// TIA Portal project "Aufgabe_2_001_mCopilot" (V20)

(* hardware
DEVICE "S7-1200 G2 station_1"  S7-1200 G2 Station
   slot 0: "Rack_0"  S71200G2 Rack  Rack  V1.0
   slot 1: "PLC_1"  CPU 1212C DC/DC/DC  6ES7 212-1AG50-0XB0  V1.0
*)

// ===== PLC "PLC_1"  CPU 1212C DC/DC/DC =====

VAR_GLOBAL   // PLC tag table "Default tag table"
   "S1" AT %I0.0 : Bool;
   "S2" AT %I0.1 : Bool;
   "S3" AT %I0.2 : Bool;
   "S4" AT %I0.3 : Bool;
   "M1" AT %Q0.0 : Bool;
   "M2" AT %Q0.1 : Bool;
   "M3" AT %Q0.2 : Bool;
   "M4" AT %Q0.3 : Bool;
   "Clock_Byte" AT %MB0 : Byte;
   "Clock_10Hz" AT %M0.0 : Bool;
   "Clock_5Hz" AT %M0.1 : Bool;
   "Clock_2.5Hz" AT %M0.2 : Bool;
   "Clock_2Hz" AT %M0.3 : Bool;
   "Clock_1.25Hz" AT %M0.4 : Bool;
   "Clock_1Hz" AT %M0.5 : Bool;
   "Clock_0.625Hz" AT %M0.6 : Bool;
   "Clock_0.5Hz" AT %M0.7 : Bool;
   "VarOverflow" AT %Q0.4 : Bool;
END_VAR

VAR_GLOBAL CONSTANT   // PLC tag table "Default tag table"
   "WARNING_THRESHOLD" : Int := 100;
END_VAR

// folder: Instances

DATA_BLOCK "InstFB_BaggageCarousel"   // DB1
{ S7_Optimized_Access := 'TRUE' }
VERSION : 0.1
// stored: InstanceOfName FB_BaggageCarousel
"FB_BaggageCarousel"
BEGIN
END_DATA_BLOCK

// folder: System blocks/Program resources

DATA_BLOCK "InstTickCunt"   // DB2
{ S7_Optimized_Access := 'TRUE' }
AUTHOR : SIMATIC
FAMILY : IEC
NAME : DCNTR
VERSION : 1.2
// stored: InstanceOfName IEC_DCOUNTER
"IEC_DCOUNTER"
BEGIN
END_DATA_BLOCK

// folder: (top level)

FUNCTION_BLOCK "FB_BaggageCarousel"   // FB21, SCL
{ S7_Optimized_Access := 'TRUE' }
VERSION : 0.1
   VAR_INPUT
      infeedConveyorS1 : Bool;   // S1
      infeedConveyorS2 : Bool;   // S2
      infeedConveyorS3 : Bool;   // S3
      circularConveyorS4 : Bool;   // S4
      clockInput : DInt;
   END_VAR
   VAR_OUTPUT
      infeedCoveyorM1 : Bool;   // M1
      infeedCoveyorM2 : Bool;   // M2
      infeedCoveyorM3 : Bool;   // M3
      circularConveyorM4 : Bool;   // M4
      clockReset : Bool;
   END_VAR
   VAR
      statInfeedConveyorM3Run : Bool;
      statInfeedConveyorM2Run : Bool;
      statInfeedConveyorM1Run : Bool;
      instInfeedPointAllowWindow : TP_TIME;
      instInfeedPointMonitor : TON_TIME;
      statClockMem : Array[0..100] of DInt;
      statClockCurrent : DInt;
      statInfeedConveyorS1BaggageDetected : Bool;   // S1
      statInfeedConveyorS2BaggageDetected : Bool;   // S2
      statInfeedConveyorS3BaggageDetected : Bool;   // S3
      statCircularConveyorS4BaggageDetectedOld : Bool;
      statSaveClock : Bool;
      statClearClockMem : Bool;
      statClockMemIndex : Int;
      statRequest : Int;
      statLoadClock : Bool;
      statLoadedClockValue : DInt;
      statIndex : Int;
      instCircularConveyorS4Monitoring : TON_TIME;   // S4 monitoring
      "instInfeed#3RequestTransferInterval" : TON_TIME;   // Interval of Infeed #3 request transfer
      instInfeedConveyorS3Off : F_TRIG;   // S3 off capture
      statInfeedConveyorM3HandleStep : Int;
      instFIFO : "FB_FIFO";
   END_VAR
   VAR_TEMP
      tempIndex : Int;
   END_VAR
   VAR CONSTANT
      ALLOW_RUN : Bool := TRUE;
      GENERALDELAY : Time := T#3000ms;
   END_VAR
BEGIN
   REGION BLOCK INFO HEADER
       //===============================================================================
       //-------------------------------------------------------------------------------
       // Title:            FB_BaggageCarousel
       // Comment/Function: This Block represents how to control the bagggage carousel which consisit of an outer circular conveyor belt (driven by M4) and
       //                   a 3-segment linear infeed conveyor belt (driven by M1, M2 & M3) based on the feedback of the corresponding baggage detection sensors S1 ~ S4.
       // Library/Family:   N.A
       // Author:           ---
       // Tested with:      S7-1200 G2/CPU 1212C DC/DC/DC FW 1.0 
       // Engineering:      TIA Portal V20
       // Requirements:     --- 
       //-------------------------------------------------------------------------------
       // Change log table:
       // Version  | Date       | Expert in charge        | Changes applied
       //----------|------------|-------------------------|-----------------------------
       // 01.00.00 | 15.12.2025 |          N.N            | First released version
       //===============================================================================
   END_REGION BLOCK INFO HEADER

   REGION DESCRIPTION  
       (/*This FB is used to control a baggage carousel system which consists of two main components: 
   A circular conveyor belt (the main conveyor) and a 3-segment linear infeed conveyor belt (for feeding baggage to main conveyor).
   - Circular conveyor belt M4 is running stable at 3.78 km/h in anticlockwise direction. Sensor S4 is equipped on it to detect the baggage
      and located near the infeed conveyor.
   - Infeed conveyor belt M1 and M2 will run accordingly to the status of subsequent infeed conveyor. Sensor S1 and S2 is equipped on 
     M1 and M2 to detect the baggage.
   - A global clock is counting. When S4 is triggered, the current clock value will be saved for the following calculation.
   - The running timing of infeed conveyor belt M3 will be calculated to avoid baggage collision in infeed area of two conveyor belts. 
     Sensor S3 is equipped on it for baggage detection. When S3 is triggered, the first saved clock will be loaded for calculation.*/)

   END_REGION DESCRIPTION

   REGION INPUT
       #statClockCurrent := #clockInput;
       #"statInfeedConveyorS1BaggageDetected" := #"infeedConveyorS1";
       #"statInfeedConveyorS2BaggageDetected" := #"infeedConveyorS2";
       #"statInfeedConveyorS3BaggageDetected" := #"infeedConveyorS3";
       IF #circularConveyorS4 AND #circularConveyorS4 <> #statCircularConveyorS4BaggageDetectedOld THEN
           #statSaveClock := TRUE;
       END_IF;
       #statCircularConveyorS4BaggageDetectedOld := #circularConveyorS4;
       #"instCircularConveyorS4Monitoring"(IN := NOT #circularConveyorS4, PT := t#11s);
       IF #"instCircularConveyorS4Monitoring".Q AND #statClockMemIndex > 0 THEN
           #statClearClockMem := TRUE;
       END_IF;
   END_REGION INPUT

   REGION PROCESSING
       #"statInfeedConveyorM1Run" := NOT (NOT #"statInfeedConveyorM2Run" AND #"statInfeedConveyorS1BaggageDetected");
       #"statInfeedConveyorM2Run" := NOT (NOT #"statInfeedConveyorM3Run" AND #"statInfeedConveyorS2BaggageDetected");
       IF NOT #"statInfeedConveyorS3BaggageDetected" THEN
           #"statInfeedConveyorM3Run" := TRUE;
       ELSE
           CASE #statInfeedConveyorM3HandleStep OF
               0:
                   IF #"statInfeedConveyorS3BaggageDetected" THEN
                       IF #statLoadedClockValue > 0 THEN
                           #statInfeedConveyorM3HandleStep := 1;
                           #statRequest += 1;
                       ELSE
                           IF #statClockMemIndex > 0 THEN
                               #statInfeedConveyorM3HandleStep := 1;
                               #statRequest += 1;
                           ELSE
                               #"statInfeedConveyorM3Run" := TRUE;
                           END_IF;
                       END_IF;
                   END_IF;
               1:
                   IF #statLoadedClockValue + 5 < #statClockCurrent AND #statLoadedClockValue + 10 > #statClockCurrent THEN
                       #"statInfeedConveyorM3Run" := FALSE;
                       #statInfeedConveyorM3HandleStep := 2;
                   END_IF;
                   IF #statLoadedClockValue + 5 >= #statClockCurrent THEN
                       #"statInfeedConveyorM3Run" := TRUE;
                       #statInfeedConveyorM3HandleStep := 4;
                   END_IF;
                   IF #statLoadedClockValue + 10 < #statClockCurrent THEN
                       #"statInfeedConveyorM3Run" := FALSE;
                       #statInfeedConveyorM3HandleStep := 3;
                   END_IF;
               2:
                   IF #"instInfeed#3RequestTransferInterval".Q THEN
                       #statInfeedConveyorM3HandleStep := 3;
                   END_IF;
               3:
                   #statInfeedConveyorM3HandleStep := 0;
                   #statLoadClock := TRUE;
           END_CASE;
       END_IF;
       #"instInfeedConveyorS3Off"(CLK := #"statInfeedConveyorS3BaggageDetected");
       IF #"instInfeedConveyorS3Off".Q THEN
           #statRequest := 0;
           #statInfeedConveyorM3HandleStep := 0;
       END_IF;
       #"instInfeed#3RequestTransferInterval"(IN := #statInfeedConveyorM3HandleStep = 2, PT := T#3000ms);

       //When 'store' is true, the below FB will store current clock into 'clockMem' array.
       //When 'load' is true, the below FB will load the value of first index of 'clockMem' array and send it to output 'loadedClockValue'.
       //The current index of 'clockMem' array is counted.
       #instFIFO(clockCurrent:=#statClockCurrent,
                 loadedClockValue=>#statLoadedClockValue,
                 clockMemIndex=>#statClockMemIndex,
                 save:=#statSaveClock,
                 load:=#statLoadClock,
                 clear:=#statClearClockMem,
                 clockMem:=#statClockMem);

   END_REGION PROCESSING

   REGION OUTPUT
       #"infeedCoveyorM1" := #"statInfeedConveyorM1Run";
       #"infeedCoveyorM2" := #"statInfeedConveyorM2Run";
       #"infeedCoveyorM3" := #"statInfeedConveyorM3Run";
       #circularConveyorM4 := TRUE;
   END_REGION OUTPUT
END_FUNCTION_BLOCK

FUNCTION "FC_Check" : Void   // FC1, SCL
{ S7_Optimized_Access := 'TRUE' }
VERSION : 0.1
BEGIN
   //Funktionsinhalt nur zur Ueberpruefung der korrekten Verknuepfung des Projekts,
   //mit dem Engineering Copilot
   //
   //Rechenaufgabe
   //Berechne die Summe von 6 und 3
END_FUNCTION

ORGANIZATION_BLOCK "Main"   // OB1, LAD, ProgramCycle
TITLE = "Main Program Sweep (Cycle)"
{ S7_Optimized_Access := 'TRUE' }
VERSION : 0.1
   VAR_INPUT
      Initial_Call : Bool;   // Initial call of this OB
      Remanence : Bool;   // =True, if remanent data are available
   END_VAR
BEGIN

REGION Network 1: SCL Comprehension
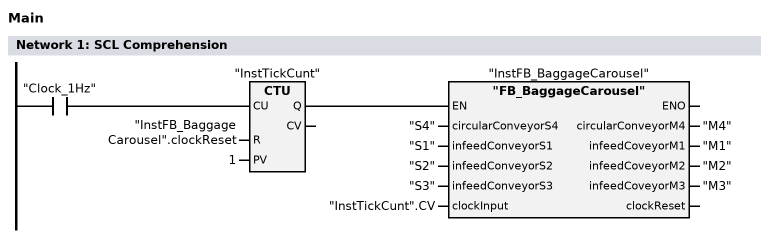
   "InstTickCunt".CTU(CU := "Clock_1Hz", R := "InstFB_BaggageCarousel".clockReset, PV := 1);
   IF "InstTickCunt".Q THEN
       "InstFB_BaggageCarousel"(circularConveyorS4 := "S4",   // "FB_BaggageCarousel"
                               infeedConveyorS1 := "S1",
                               infeedConveyorS2 := "S2",
                               infeedConveyorS3 := "S3",
                               clockInput := "InstTickCunt".CV,
                               circularConveyorM4 => "M4",
                               infeedCoveyorM1 => "M1",
                               infeedCoveyorM2 => "M2",
                               infeedCoveyorM3 => "M3");
   END_IF;
END_REGION
END_ORGANIZATION_BLOCK

// folder: BasicFunction

FUNCTION_BLOCK "FB_FIFO"   // FB100, SCL
{ S7_Optimized_Access := 'TRUE' }
VERSION : 0.1
   VAR_INPUT
      clockCurrent : DInt;
   END_VAR
   VAR_OUTPUT
      loadedClockValue : DInt;
      clockMemIndex : Int;
   END_VAR
   VAR_IN_OUT
      save : Bool;
      load : Bool;
      clear : Bool;
      clockMem : Array[*] of DInt;
   END_VAR
   VAR
      statIndex : Int;
      statUpperBound : DInt;
      statLowerBound : DInt;
   END_VAR
   VAR_TEMP
      tempIndex : Int;
   END_VAR
BEGIN
   REGION FIFO
       #statLowerBound := LOWER_BOUND(ARR := #clockMem, DIM := 1);
       #statUpperBound := UPPER_BOUND(ARR := #clockMem, DIM := 1);
       IF #save THEN
           #clockMem[#statIndex] := #clockCurrent;
           #save := FALSE;
           #statIndex += 1;
       END_IF;
       IF #load THEN
           IF #statIndex > 0 THEN
               #loadedClockValue := #clockMem[#statLowerBound];
               FOR #tempIndex := #statLowerBound TO #statIndex - 1 DO
                   #clockMem[#tempIndex] := #clockMem[#tempIndex + 1];
               END_FOR;
               #statIndex -= 1;
           ELSE
               #loadedClockValue := 0;
           END_IF;
           #load := FALSE;
       END_IF;
       IF #clear THEN
           FOR #tempIndex := #statLowerBound TO #statUpperBound DO
               #clockMem[#tempIndex] := 0;
           END_FOR;
           #clear := FALSE;
           #loadedClockValue := 0;
           #statIndex := 0;
       END_IF;
       IF #statIndex = #statUpperBound THEN
           #statIndex := DINT_TO_INT(#statLowerBound);
       END_IF;
       #clockMemIndex := #statIndex;
   END_REGION FIFO
END_FUNCTION_BLOCK

// ===== library types =====

// folder: LGF/7 Signal generators

FUNCTION_BLOCK "LGF_Frequency"   // FB10024, SCL
TITLE = LGF_Frequency
{ S7_Optimized_Access := 'TRUE' }
AUTHOR : Siemens_Industry_Support
FAMILY : LGF
NAME : LGF_Frequency
// This function generates a signal that changes between the values `FALSE` and `TRUE` depending on a defined frequency and a pulse pause ratio. / Diese Funktion generiert ein Signal, das in Abhängigkeit von einer definierten Frequenz und einem Pulspausenverhältnis, zwischen den Werten `FALSE` und `TRUE` wechselt.
   VAR_INPUT
      frequency : Real := 0.0;   // Clock frequency in Hz. / Taktfrequenz in Hz.
      pulsePauseRatio : Real := 1.0;   // Pulse pause ratio (standard: 1.0 corresponds to 1:1). / Pulspausenverhältnis (Standard: 1.0 entspricht 1:1).
   END_VAR
   VAR_OUTPUT
      clock : Bool;   // Output changes with defined frequency. / Ausgang wechselt mit definierter Frequenz.
      countdown : Time;   // Remaining time of the current `clock` state. / Verbleibende Zeit des aktuellen Zustands von `clock`.
   END_VAR
   VAR
      instTofTimePulse : TOF_TIME;   // Timer instance for the Pulse signal (Period of time the clock signal is true)
      instTofTimePause : TOF_TIME;   // Timer instance for the Pause signal (Period of time the clock signal is false)
      statFrequencyOld : Real;   // Static Old/Current value of the frequency input
      statPulsePauseRatioOld : Real;   // Static Old/Current value of the pulsePauseRatio input
      statTimePulse : Time;   // Static calculated for me the pulse duration of the clock
      statTimePause : Time;   // Static calculated for me the pause duration of the clock
   END_VAR
   VAR_TEMP
      tempPulseRate : Real;   // Static calculation of pulse rate - needed for passing value between calculations
      tempPauseRate : Real;   // Static calculation of pause rate - needed for passing value between calculations
      tempCountdown : Time;   // Static countdown until next ON/OFF value of the clock signal
   END_VAR
   VAR CONSTANT
      ZERO : Real := 0.0;   // Numeric zero constant
      ZERO_TIME : Time := T#0ms;   // Time zero constant
      SECOND_IN_MS : Real := 1000.0;   // One second written in miliseconds. Needed in calculation in formulas
      ONE : Real := 1.0;   // 100% - One hundred procent / 100% - Einhundert Prozent
   END_VAR
BEGIN
   REGION Block info header
     //=============================================================================
     // SIEMENS AG / (c)Copyright 2017
     //-----------------------------------------------------------------------------
     // Title:            LGF_Frequency
     // Comment/Function: This function generates a signal that changes between the values `FALSE` and `TRUE` depending on a defined frequency and a pulse pause ratio.
     // Library/Family:   LGF(Library General Functions)
     // Author:           Siemens Digital Industry Support
     // Tested with:      S7-PLCSIM Advanced V2.0 SP1
     // Engineering:      TIA Portal V15 Update 2
     // Restrictions:     ENO disabled - error handling done by error and status
     // Requirements:     PLC (S7-1200 / S7-1500)
     //-------------------------------------------------------------------------------
     // Change log table:
     // Version  | Date       | Expert in charge       | Changes applied
     //----------|------------|------------------------|------------------------------
     // 01.00.00 19.08.2015  Siemens Industry Online Support
     //                      First released version
     // 01.01.00 25.05.2016  Siemens Industry Online Support
     //                      New function: pulse pause ratio
     // 01.01.01 26.05.2016  Siemens Industry Online Support
     //                      Add comments
     // 01.01.02 02.01.2017  Siemens Industry Online Support
     //                      Upgrade: TIA Portal V14 Update 1
     // 01.01.03 17.08.2018  Siemens Industry Online Support
     //                      Upgrade: TIA V15 Update 2
     // 01.01.04 23.11.2018  Siemens Industry Online Support
     //                      Upgrade: TIA V15.1
     // 01.00.07 20.09.2019  Simatic Systems Support
     //                      Code refactoring, regions and more comments added
     // 03.00.00 23.04.2020  Simatic Systems Support
     //                      Set version to V3.0.0, harmonize the version of the whole library
     // 03.00.01 15.02.2021  Simatic Systems Support
     //                      Insert documentation
     //=============================================================================
   END_REGION Block info header

   REGION DESCRIPTION
     (/*The `clock` output is a Boolean value that toggles at the desired frequency. The `pulsePauseRatio` input is used to set the pulse pause ratio.

   The output `countdown` outputs the remaining time of the current state of `clock`.

   If the desired frequency or pulse pause ratio is less than or equal to `0.0`, the output `clock` = FALSE and `countdown` = `0s`.

   ------

   #### Example

   ![LGF_Frequency](LGF_Frequency.png "LGF_Frequency")

   ---

   Note
   :    The `clock` of the FB LGF_Frequency depends on the cycle time of the OB
   Main. To increase the accuracy, the FB can also be called in a cyclic interrupt
   OB with a low time interval.
   Der Ausgang `clock` ist ein boolescher Wert, der in der gewünschten Frequenz toggelt. Über den Eingang `pulsePauseRatio` wird das Pulspausenverhältnis eingestellt.

   Der Ausgang `countdown` gibt die verbleibende Zeit des aktuellen Zustands von `clock` aus.

   Falls die gewünschte Frequenz oder das Pulspausenverhältnis kleiner oder gleich `0.0` ist, ist der Ausgang `clock` = FALSE und `countdown` = `0s`.

   ------

   #### Beispiel

   ![LGF_Frequency](LGF_Frequency.png "LGF_Frequency")

   ---

   Hinweis
   :    Der Takt (`clock`) des FB LGF_Frequency ist abhängig von der Zykluszeit des OB Main. Um die Genauigkeit zu erhöhen, kann der FB auch in einem Weckalarm-OB (Cyclic Interrupt OB) mit niedrigem Zeittakt aufgerufen werden.*/)
   END_REGION DESCRIPTION

   REGION Calculation of settings and program execution
     // If input <= 0.0 the block is disabled
     IF (#frequency <= #ZERO) OR (#pulsePauseRatio <= #ZERO) THEN
       #clock := FALSE;
       #tempCountdown := #ZERO_TIME;
     ELSE

       //Calculating function frequency and pulse pause ratio only when an input is changed
       IF #statFrequencyOld <> #frequency OR #statPulsePauseRatioOld <> #pulsePauseRatio THEN
         RESET_TIMER(TIMER := #instTofTimePause);
         RESET_TIMER(TIMER := #instTofTimePulse);

         #tempPulseRate := #pulsePauseRatio / (#pulsePauseRatio + #ONE); // Calculate pulse rate   
         #tempPauseRate := #ONE - #tempPulseRate;                      // Calculate pause rate   
         #statTimePulse := UDINT_TO_TIME(REAL_TO_UDINT((#SECOND_IN_MS * #tempPulseRate / #frequency))); // Calculate pulse time   
         #statTimePause := UDINT_TO_TIME(REAL_TO_UDINT((#SECOND_IN_MS * #tempPauseRate / #frequency))); // Calculate pause time
         #statFrequencyOld := #frequency;
         #statPulsePauseRatioOld := #pulsePauseRatio;
       END_IF;

       //Two time off-delay timers that are resetting each other on expiration
       #instTofTimePulse(IN := NOT #instTofTimePause.Q,
                         PT := #statTimePulse);

       //If timer for pulse is running, remaining time of the PULSE is calculated
       #tempCountdown := #statTimePulse - #instTofTimePulse.ET;

       #instTofTimePause(IN := #instTofTimePulse.Q,
                         PT := #statTimePause);

       //If timer for pulse is NOT running, remaining time of the PAUSE is calculated
       IF #tempCountdown = #ZERO_TIME THEN
         #tempCountdown := #statTimePause - #instTofTimePause.ET;
       END_IF;

     END_IF;
   END_REGION

   REGION Writing to outputs
     // Assigning value of the pulse timer to the clock output
     #clock := #instTofTimePulse.Q;
     #countdown := #tempCountdown;
     //ENO mechanism is not used - forced to true.
     ENO := TRUE;
   END_REGION
END_FUNCTION_BLOCK